{attribute 'qualified_only'}
VAR_GLOBAL
	fbTestsuites:			FB_Testsuites;	
END_VAR

(* stored: Version 1.1.0.1, ProductVersion 3.1.4024.12
   GVL TestSuiteGVL: Id {33e8e116-cffd-48af-9b67-4029ebba997a} *)
